Fanuc KAREL source: kc00060.KL

-- PROVISIONAL review KL for V940-1; original PC SHA256 65c7541a9b554fd866f089d1fc668e57251ba30435d0615eb4dd2a4f4e2aaa35
-- Incomplete behavior may be omitted. Consult companion uncertainty JSON. Do not deploy.
PROGRAM KC00060
%NOLOCKGROUP
BEGIN
  -- V9_ZERO_TABLE_METADATA_HINT layout=0002_ascii; no indexed target words; source/name/runtime held
  -- UNRESOLVED_PC offsets 5-43; opcodes 27,27,9D,22,1C,22,22,2A,AA,23
  -- UNRESOLVED_PC offsets 48-52; opcodes 7F
END KC00060
